DATA_BLOCK "dbArchiveParOven"
{ S7_Optimized_Access := 'TRUE' }
VERSION : 0.8
"fbArchiveParOven"

BEGIN

END_DATA_BLOCK

